TEXTLIST TextList_Config_Evap
  0 = 'reg quartz' | FR: 'Réglage quartz' | EN: 'Crystal setting'
  1 = 'life seuil' | FR: "Seuil d'alarme vie des quartz" | EN: 'Crystal life alarm threshold'
  2 = 'evap settings' | FR: 'Réglages surveillance temps maximum de dépôt' | EN: 'Maximum evaporation time monitoring settings'
  3 = 'prm_tim_surv_dep_min' | FR: 'Temps maximum définissant un dépôt court\nTemps ajouté au temps théorique pour les dépôts courts' | EN: 'Maximum time to determinate a short deposit\nTheorical additional time for short deposit'
  4 = 'PRM_Fact_Surv_Dep' | FR: 'Pourcentage temps supplémentaire ajouté pour les dépôts longs' | EN: 'Additional time porcentage for long deposit'
  5 = 'reg source 1' | FR: 'Réglages source 1' | EN: 'Source 1 settings'
  6 = 'reg source 2' | FR: 'Réglages source 2' | EN: 'Source 2 settings'
  7 = 'matériau' | FR: 'Matériau' | EN: 'Material'
  8 = 'Nom balayage' | FR: 'Nom du balayage' | EN: 'Sweeping name'
  9 = 'no mvts in proc' | FR: 'Inhibition des mouvements canne en process' | EN: 'No transfer arm movements in process'
  10 = 'reglages mvts' | FR: 'Réglages mouvements' | EN: 'Movement settings'
  11 = 'evap continue' | FR: 'Mode évaporation continue' | EN: 'Continuous evaporation mode'
  12 = 'mode actif' | FR: 'Mode évaporation continue actif (si non, mode couche classique)' | EN: 'Continuous evaporation mode active (if not, classical layer mode)'
  13 = 'rate watcher time' | FR: "Interval de temps entre les périodes d'échantillonage" | EN: 'Time interval between sample periods'
  14 = 'rate watcher accuracy' | FR: "Tolérance de la fenêtre de validation de la vitesse d'évaporation" | EN: 'Acceptance window for evaporation rate'
  15 = 'maximum time' | FR: "Temps maximum d'évaporation continue avant arrêt automatique" | EN: 'Maximum time for continuous evaporation before automatic stop'
  16 = 'confirm refill' | FR: 'Cliquez ici pour confirmer que les creusets ont été chargés' | EN: 'Click here to confirm crucible refilling'
  17 = 'maximum time s1' | FR: "Temps maximum d'évaporation continue avant arrêt automatique (Canon 1)" | EN: 'Maximum time for continuous evaporation before automatic stop (E-Gun 1)'
  18 = 'maximum time s2' | FR: "Temps maximum d'évaporation continue avant arrêt automatique (Source Joule)" | EN: 'Maximum time for continuous evaporation before automatic stop (Thermal source)'
  19 = 'maximum time s3' | FR: "Temps maximum d'évaporation continue avant arrêt automatique (Canon 2)" | EN: 'Maximum time for continuous evaporation before automatic stop (E-Gun 2)'
  20 = 'Reg XTC' | FR: 'Réglage XTC' | EN: 'XTC Setting'
  21 = 'IP' | FR: "Adresse IP de l'XTC" | EN: 'Ip Adress of XTC'
  22 = 'Cr' | FR: 'Creuset' | EN: 'Crucible'
  23 = 'CONF_Min_Temp_IN' | FR: 'Température min. eau en entrée du canon' | EN: 'Min. water temperature at gun inlet'
  24 = 'CONF_Max_Temp_IN' | FR: 'Température max. eau en entrée du canon' | EN: 'Max. water temperature at gun inlet'
  25 = 'CONF_Min_Temp_OUT' | FR: 'Température min. eau en sortie du canon' | EN: 'Min. water temperature at gun outlet'
  26 = 'CONF_Max_Temp_OUT' | FR: 'Température max. eau en sortie du canon' | EN: 'Max. water temperature at gun outlet'
  27 = 'reg eau' | FR: 'Réglages température eau' | EN: 'Water temperature settings'
   = ''
END_TEXTLIST

(* stored: Version 1.1.0.1, ProductVersion 3.1.4024.12
   TextList TextList_Config_Evap: Id {94edaa7a-b0b7-43bc-af1e-724a121088c2} *)
